# EPICS StreamDevice protocol: device.proto
# =========================================================
# StreamDevice Protocol File
# =========================================================

Terminator = LF;

# =========================================================
# READ TEMPERATURE
# =========================================================

getValue {
    out "TEMP?";
    in "%f";
}
